FUNCTION_BLOCK FB_PowerNC IMPLEMENTS I_Power
VAR_INPUT
END_VAR
VAR_OUTPUT
END_VAR
VAR
    {attribute 'no_copy'}
    AxisRef : REFERENCE TO AXIS_REF;
    fbMcPower : MC_Power;
    bEnable	: BOOL;
    bEnablePositive : BOOL;
    bEnableNegative : BOOL;
    bPowerIsEnabled : BOOL;
    bBusy 		: BOOL;
    bError 	: BOOL;
    nErrorID 	: UDINT;
    fOverride 	: LREAL := 100.0;
    eBufferMode : MC_BufferMode := MC_BufferMode.MC_Aborting;
END_VAR

//////////////////////////////////////////////////////////////////
// Power block depends on interlocks check in  iMotionInterlocks
/////////////////////////////////////////////////////////////////
THIS^.fbMcPower(
    Axis := THIS^.AxisRef,
    Enable := THIS^.bEnable,
    Enable_Positive := THIS^.bEnablePositive,
    Enable_Negative := THIS^.bEnableNegative,
    Override := THIS^.fOverride,
    BufferMode := THIS^.eBufferMode,
    (*Enabled*)
    Status => THIS^.bPowerIsEnabled,
    Busy => THIS^.bBusy,
    Error => THIS^.bError,
    ErrorID => THIS^.nErrorID
);

//FB_Init is always available implicitly and it is used primarily for initialization.
//The return value is not evaluated. For a specific influence, you can also declare the
//methods explicitly and provide additional code there with the standard initialization
//code. You can evaluate the return value.
METHOD FB_Init: BOOL
VAR_INPUT
    bInitRetains: BOOL; // TRUE: the retain variables are initialized (reset warm / reset cold)
    bInCopyCode: BOOL;  // TRUE: the instance will be copied to the copy code afterward (online change)
    AxisRef : REFERENCE TO AXIS_REF;
END_VAR
THIS^.AxisRef REF= AxisRef;
END_METHOD

METHOD Power
VAR_INPUT
    Enable	: BOOL;
    Enable_Positive	: BOOL;
    Enable_Negative	: BOOL;
    (* in percent from 0 to 100 *)
    Override	: LREAL := 100;
    BufferMode	: MC_BufferMode := .MC_BufferMode.MC_Aborting;
END_VAR
THIS^.bEnable := Enable;
THIS^.bEnablePositive := Enable_Positive;
THIS^.bEnableNegative := Enable_Negative;
THIS^.fOverride := Override;
THIS^.eBufferMode := BufferMode ;
END_METHOD

{warning 'Add property implementation'}
PROPERTY PowerActive : BOOL
GET
END_GET
END_PROPERTY

METHOD PowerEnables
VAR_INPUT
    Enable	: BOOL;
    Enable_Positive	: BOOL;
    Enable_Negative	: BOOL;
END_VAR
THIS^.bEnable := Enable;
THIS^.bEnablePositive := Enable_Positive;
THIS^.bEnableNegative := Enable_Negative;
END_METHOD

{warning 'add property implementation'}
PROPERTY PowerError : BOOL
GET
PowerError := bError;
END_GET
END_PROPERTY

PROPERTY PowerErrorID : UDINT
GET
PowerErrorID := nErrorID;
END_GET
END_PROPERTY

{attribute 'monitoring':= 'variable'}
PROPERTY PowerIsEnabled : BOOL
GET
PowerIsEnabled := bPowerIsEnabled;
END_GET
END_PROPERTY

END_FUNCTION_BLOCK

(* stored: Version 1.1.0.1
   POU FB_PowerNC: Id {82bac45d-f3fb-4090-96f5-9cec57f017c8}, SpecialFunc None
   Method FB_Init: Id {cf7caa46-f1e4-49f9-addf-eba93ec02164}
   Method Power: Id {b859403c-f315-4c59-bb46-554245f47326}
   Property PowerActive: Id {49693f07-c88b-4b06-be0c-0dc75c8f5fac}
   Get Get: Id {b11a8d39-0dfc-40d5-ab4e-e7fe1f8bda7c}
   Method PowerEnables: Id {60dea20e-362a-45d5-ab02-9c322c575503}
   Property PowerError: Id {5900c701-bb24-4682-9d2c-47b8d2773b46}
   Get Get: Id {50fb1906-033c-485b-9e5d-f1230f94dfc8}
   Property PowerErrorID: Id {1fe914ad-7f24-41a0-bde2-d4d693aeb73f}
   Get Get: Id {8f8eef06-c2be-4844-866a-ef0542739cd8}
   Property PowerIsEnabled: Id {7e136934-4440-48f5-a211-011704d8f4f5}
   Get Get: Id {fffb35ff-b9f5-44f8-bd6c-842b697893c4} *)
